{attribute 'qualified_only'}
VAR_GLOBAL
END_VAR

(* stored: Version 1.1.0.1, ProductVersion 3.1.4022.7
   GVL GVL_07_Alarm_Servo_Motor_Shelf_Y: Id {f4dbec09-073e-4d3a-af86-11f55bd6ac1c} *)
